Staubli VAL3: stop.pgx

program stop()
begin
  waitEndMove()
  cls()
  title("")
  gotoxy(17,7)
  putln("-END-")
  resetMotion()
end
